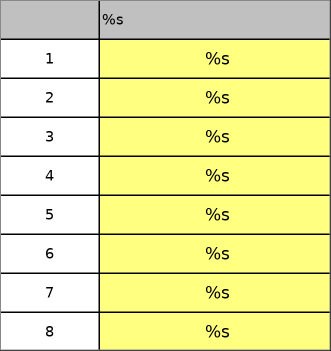
VISUALIZATION VISU_CONF_MAT  // 331x351
VAR_IN_OUT
	m_Input_CRUCIBLE : BLOCK_IND_CR_396_TELEMARK;
END_VAR
    Rectangle (0,0 99x39)
    Rectangle (99,39 232x39), "%s", text variable: m_Input_CRUCIBLE.PRM_MAT[1], input disabled if: NOT Global_Variables.PRG_USER.ACTU_USER.CONF_MACHINE
        OnMouseDown: write the text variable via InputWithLimits
    Rectangle (99,0 232x39), "%s", text list: 'TextList_Config_Evap', text index: 7
    Rectangle (0,39 99x39), "1"
    Rectangle (0,78 99x39), "2", invisible if: m_Input_CRUCIBLE.CONF_NCR <2
    Rectangle (99,78 232x39), "%s", text variable: m_Input_CRUCIBLE.PRM_MAT[2], invisible if: m_Input_CRUCIBLE.CONF_NCR <2, input disabled if: NOT Global_Variables.PRG_USER.ACTU_USER.CONF_MACHINE
        OnMouseDown: write the text variable via InputWithLimits
    Rectangle (0,117 99x39), "3", invisible if: m_Input_CRUCIBLE.CONF_NCR <3
    Rectangle (99,117 232x39), "%s", text variable: m_Input_CRUCIBLE.PRM_MAT[3], invisible if: m_Input_CRUCIBLE.CONF_NCR <3, input disabled if: NOT Global_Variables.PRG_USER.ACTU_USER.CONF_MACHINE
        OnMouseDown: write the text variable via InputWithLimits
    Rectangle (0,156 99x39), "4", invisible if: m_Input_CRUCIBLE.CONF_NCR <4
    Rectangle (99,156 232x39), "%s", text variable: m_Input_CRUCIBLE.PRM_MAT[4], invisible if: m_Input_CRUCIBLE.CONF_NCR <4, input disabled if: NOT Global_Variables.PRG_USER.ACTU_USER.CONF_MACHINE
        OnMouseDown: write the text variable via InputWithLimits
    Rectangle (0,195 99x39), "5", invisible if: m_Input_CRUCIBLE.CONF_NCR <5
    Rectangle (99,195 232x39), "%s", text variable: m_Input_CRUCIBLE.PRM_MAT[5], invisible if: m_Input_CRUCIBLE.CONF_NCR <5, input disabled if: NOT Global_Variables.PRG_USER.ACTU_USER.CONF_MACHINE
        OnMouseDown: write the text variable via InputWithLimits
    Rectangle (0,234 99x39), "6", invisible if: m_Input_CRUCIBLE.CONF_NCR <6
    Rectangle (99,234 232x39), "%s", text variable: m_Input_CRUCIBLE.PRM_MAT[6], invisible if: m_Input_CRUCIBLE.CONF_NCR <6, input disabled if: NOT Global_Variables.PRG_USER.ACTU_USER.CONF_MACHINE
        OnMouseDown: write the text variable via InputWithLimits
    Rectangle (0,273 99x39), "7", invisible if: m_Input_CRUCIBLE.CONF_NCR <7
    Rectangle (99,273 232x39), "%s", text variable: m_Input_CRUCIBLE.PRM_MAT[7], invisible if: m_Input_CRUCIBLE.CONF_NCR <7, input disabled if: NOT Global_Variables.PRG_USER.ACTU_USER.CONF_MACHINE
        OnMouseDown: write the text variable via InputWithLimits
    Rectangle (0,312 99x39), "8", invisible if: m_Input_CRUCIBLE.CONF_NCR <8
    Rectangle (99,312 232x39), "%s", text variable: m_Input_CRUCIBLE.PRM_MAT[8], invisible if: m_Input_CRUCIBLE.CONF_NCR <8, input disabled if: NOT Global_Variables.PRG_USER.ACTU_USER.CONF_MACHINE
        OnMouseDown: write the text variable via InputWithLimits
END_VISUALIZATION

(* stored: Version 1.1.0.1, ProductVersion 3.1.4026.18
   Visu VISU_CONF_MAT: Id {98f4d72d-5ad7-4275-9f39-1bb9579ecc17} *)
